TYPE MultiAxis_Status_typ :
	STRUCT
		Done  		: BOOL;
		Busy 		: BOOL;
	END_STRUCT
END_TYPE

(* stored: Version 1.1.0.1, ProductVersion 3.1.4024.3
   DUT MultiAxis_Status_typ: Id {104efeec-b799-086b-07e1-57cb93520783} *)
